KUKA KRL data list: KukaMatlabConnection_min.dat

&ACCESS RVP
&REL 57
&PARAM TEMPLATE = C:\KRC\Roboter\Template\vorgabe
&PARAM EDITMASK = *
DEFDAT KukaMatlabConnection

EXT  BAS (BAS_COMMAND  :IN,REAL  :IN )
DECL INT SUCCESS

DECL RSIERR err
INT hEthernet
INT hAxis,hPath
INT UNIT_RSI

ENDDAT
